FUNCTION_BLOCK Test_ExampleTest EXTENDS T_UnitTestBase IMPLEMENTS I_UnitTest
VAR_INPUT
END_VAR
VAR_OUTPUT
END_VAR
VAR
	TestByte : BYTE := 123;
END_VAR

Assertion.AssertEquals_BYTE(Expected     := 123,
                            Actual       := TestByte,
                            VariableName := 'TestByte');

CheckAssertion(NextState := 0);

END_FUNCTION_BLOCK

(* stored: Version 1.1.0.1, ProductVersion 3.1.4024.11
   POU Test_ExampleTest: Id {154b81fb-5e29-4f42-a15a-b536fe2b7a5c}, SpecialFunc None *)
